TYPE Cnv_Level_Settings_DUT :
STRUCT
	Cnv1:	Buffer_Cnv_Settings_DUT;
	Cnv2:	Buffer_Cnv_Settings_DUT;
END_STRUCT
END_TYPE

(* stored: Version 1.1.0.1
   DUT Cnv_Level_Settings_DUT: Id {d3365a0d-bea5-495e-8398-a920b8ff764a} *)
